// TIA Portal project "durum_grafigi_2_asansor" (V18)

(* hardware
DEVICE "S7-1200 station_1"  S7-1200 Station
   slot 0: "Rack_0"  S7-1200 Rack  Rack  V1.0
   slot 1: "PLC_1"  CPU 1214C DC/DC/DC  6ES7 214-1AG40-0XB0  V4.6
*)

// ===== PLC "PLC_1"  CPU 1214C DC/DC/DC =====

VAR_GLOBAL   // PLC tag table "Default tag table"
   "STOP-S0" AT %I0.0 : Bool;
   "START-S1" AT %I0.1 : Bool;
   "SAYMA SENSÖRÜ-S3" AT %I0.2 : Bool;
   "ASANSÖR AŞAĞIDA-S4" AT %I0.3 : Bool;
   "ASANSÖR YUKARIDA-S5" AT %I0.4 : Bool;
   "BANT MOTORU-M1" AT %Q0.0 : Bool;
   "ASANSÖR YUKARI-M2Y" AT %Q0.1 : Bool;
   "ASANSÖR AŞAĞI -M2A" AT %Q0.2 : Bool;
   "ASANSÖR KİLİTLEME" AT %Q0.3 : Bool;
   "PARÇA SÜRME" AT %Q0.4 : Bool;
   "DURUM_0 BAŞLANGIÇ" AT %M30.0 : Bool;
   "DURUM_1 BANT ÇALIŞTIRMA" AT %M30.1 : Bool;
   "DURUM_2 ASANSÖR YUKARI" AT %M30.2 : Bool;
   "DURUM_3 KİLİTLEME" AT %M30.3 : Bool;
   "DURUM_4 ASANSÖR AŞAĞI" AT %M30.4 : Bool;
   "System_Byte" AT %MB80 : Byte;
   "FirstScan" AT %M80.0 : Bool;
   "DiagStatusUpdate" AT %M80.1 : Bool;
   "AlwaysTRUE" AT %M80.2 : Bool;
   "AlwaysFALSE" AT %M80.3 : Bool;
   "Clock_Byte" AT %MB20 : Byte;
   "Clock_10Hz" AT %M20.0 : Bool;
   "Clock_5Hz" AT %M20.1 : Bool;
   "Clock_2.5Hz" AT %M20.2 : Bool;
   "Clock_2Hz" AT %M20.3 : Bool;
   "Clock_1.25Hz" AT %M20.4 : Bool;
   "Clock_1Hz" AT %M20.5 : Bool;
   "Clock_0.625Hz" AT %M20.6 : Bool;
   "Clock_0.5Hz" AT %M20.7 : Bool;
END_VAR

// folder: System blocks/Program resources

DATA_BLOCK "PARÇA SAYICISI"   // DB1
{ S7_Optimized_Access := 'TRUE' }
AUTHOR : Simatic
FAMILY : IEC
NAME : CNTR
VERSION : 1.0
// stored: InstanceOfName IEC_COUNTER
"IEC_COUNTER"
BEGIN
END_DATA_BLOCK

DATA_BLOCK "BEKLEME ZAMANI"   // DB2
{ S7_Optimized_Access := 'TRUE' }
AUTHOR : Simatic
FAMILY : IEC
NAME : IEC_TMR
VERSION : 1.0
// stored: InstanceOfName IEC_TIMER
"IEC_TIMER"
BEGIN
END_DATA_BLOCK

// folder: (top level)

ORGANIZATION_BLOCK "Main"   // OB1, LAD, ProgramCycle
TITLE = "Main Program Sweep (Cycle)"
{ S7_Optimized_Access := 'TRUE' }
VERSION : 0.1
// -*Asansör kabini asagida ve START butonuna basilmis ise
// bant dönmeye baslayacaktir.
// -*Bantin dönmeye baslamasiyla magazin üzerindeki
// paketler sürme silindiri yardimiyla belli araliklarla bant
// üzerine sürülecektir. Bant üzerindeki paketler SAYMA
// SENSÖRÜ önünden geçerek asansör kabinine dolacaktir.
// Kabin içerisindeki paket sayisi 5 oldugunda asansör
// yukan dogru hareket edecek ve bant duracaktir.
// -*Asansör kabini yukan çikip orada paketlerin bosalmasi
// için 5 saniye bekleyip tekrar asagi inecektir. Bekleme
// sirasinda FRENLEME çalisacaktir.
// -* START butonuna basildiginda bu islemler yeniden baslayacaktir.
// - STOP butonuna basildiginda FRENLEME çalisacak, diger motorlar duracaktir. STOP butonu
// birakildiginda BEKLEME SÜRESÌ tamamsa asansör asagi hareket edecektir.
   VAR_INPUT
      Initial_Call : Bool;   // Initial call of this OB
      Remanence : Bool;   // =True, if remanent data are available
   END_VAR
BEGIN

REGION Network 1: DURUM_0
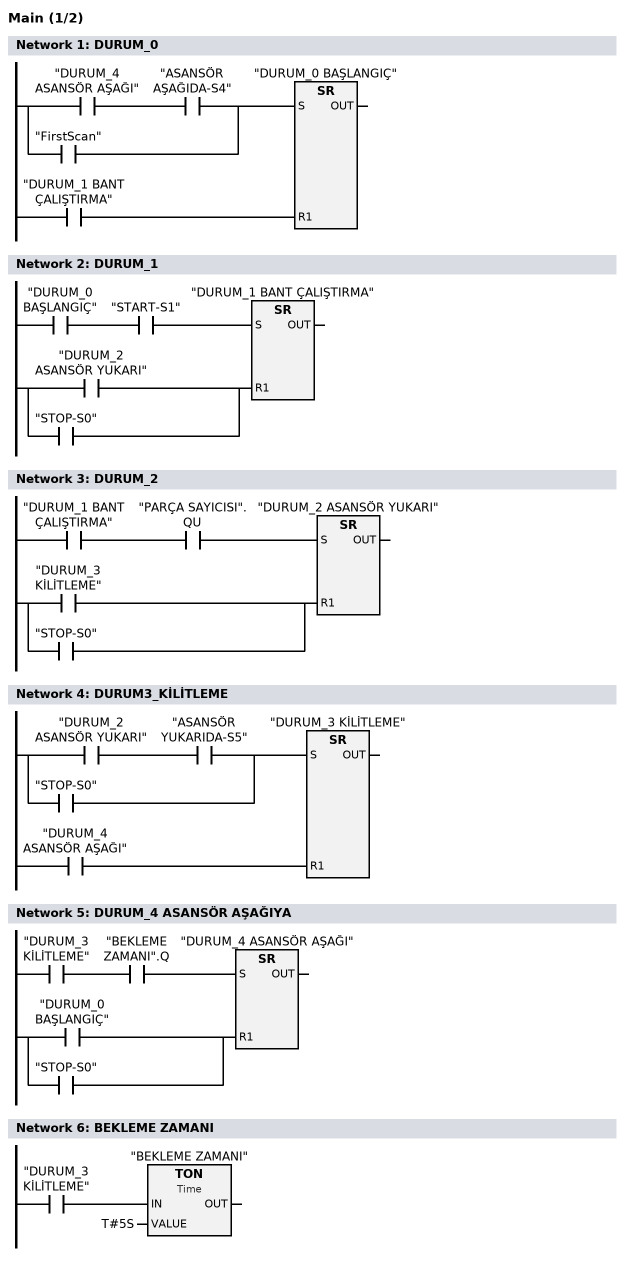
   RUNG wire#powerrail
      Contact( "DURUM_4 ASANSÖR AŞAĞI" )
      Contact( "ASANSÖR AŞAĞIDA-S4" )
      wire#w1
      S_SR(operand := "DURUM_0 BAŞLANGIÇ", r1 := wire#w2)
   END_RUNG
   RUNG wire#powerrail
      Contact( "FirstScan" )
   END_RUNG wire#w1
   RUNG wire#powerrail
      Contact( "DURUM_1 BANT ÇALIŞTIRMA" )
   END_RUNG wire#w2
   // the same network as SCL:
   IF ("DURUM_4 ASANSÖR AŞAĞI" AND "ASANSÖR AŞAĞIDA-S4") OR "FirstScan" THEN
       "DURUM_0 BAŞLANGIÇ" := TRUE;   // SR flip-flop
   END_IF;
   IF "DURUM_1 BANT ÇALIŞTIRMA" THEN "DURUM_0 BAŞLANGIÇ" := FALSE; END_IF;
END_REGION

REGION Network 2: DURUM_1
   RUNG wire#powerrail
      Contact( "DURUM_0 BAŞLANGIÇ" )
      Contact( "START-S1" )
      S_SR(operand := "DURUM_1 BANT ÇALIŞTIRMA", r1 := wire#w1)
   END_RUNG
   RUNG wire#powerrail
      Contact( "DURUM_2 ASANSÖR YUKARI" )
   END_RUNG wire#w1
   RUNG wire#powerrail
      Contact( "STOP-S0" )
   END_RUNG wire#w1
   // the same network as SCL:
   IF "DURUM_0 BAŞLANGIÇ" AND "START-S1" THEN
       "DURUM_1 BANT ÇALIŞTIRMA" := TRUE;   // SR flip-flop
   END_IF;
   IF "DURUM_2 ASANSÖR YUKARI" OR "STOP-S0" THEN "DURUM_1 BANT ÇALIŞTIRMA" := FALSE; END_IF;
END_REGION

REGION Network 3: DURUM_2
   RUNG wire#powerrail
      Contact( "DURUM_1 BANT ÇALIŞTIRMA" )
      Contact( "PARÇA SAYICISI".QU )
      S_SR(operand := "DURUM_2 ASANSÖR YUKARI", r1 := wire#w1)
   END_RUNG
   RUNG wire#powerrail
      Contact( "DURUM_3 KİLİTLEME" )
   END_RUNG wire#w1
   RUNG wire#powerrail
      Contact( "STOP-S0" )
   END_RUNG wire#w1
   // the same network as SCL:
   IF "DURUM_1 BANT ÇALIŞTIRMA" AND "PARÇA SAYICISI".QU THEN
       "DURUM_2 ASANSÖR YUKARI" := TRUE;   // SR flip-flop
   END_IF;
   IF "DURUM_3 KİLİTLEME" OR "STOP-S0" THEN "DURUM_2 ASANSÖR YUKARI" := FALSE; END_IF;
END_REGION

REGION Network 4: DURUM3_KİLİTLEME
   RUNG wire#powerrail
      Contact( "DURUM_2 ASANSÖR YUKARI" )
      Contact( "ASANSÖR YUKARIDA-S5" )
      wire#w1
      S_SR(operand := "DURUM_3 KİLİTLEME", r1 := wire#w2)
   END_RUNG
   RUNG wire#powerrail
      Contact( "STOP-S0" )
   END_RUNG wire#w1
   RUNG wire#powerrail
      Contact( "DURUM_4 ASANSÖR AŞAĞI" )
   END_RUNG wire#w2
   // the same network as SCL:
   IF ("DURUM_2 ASANSÖR YUKARI" AND "ASANSÖR YUKARIDA-S5") OR "STOP-S0" THEN
       "DURUM_3 KİLİTLEME" := TRUE;   // SR flip-flop
   END_IF;
   IF "DURUM_4 ASANSÖR AŞAĞI" THEN "DURUM_3 KİLİTLEME" := FALSE; END_IF;
END_REGION

REGION Network 5: DURUM_4 ASANSÖR AŞAĞIYA
   RUNG wire#powerrail
      Contact( "DURUM_3 KİLİTLEME" )
      Contact( "BEKLEME ZAMANI".Q )
      S_SR(operand := "DURUM_4 ASANSÖR AŞAĞI", r1 := wire#w1)
   END_RUNG
   RUNG wire#powerrail
      Contact( "DURUM_0 BAŞLANGIÇ" )
   END_RUNG wire#w1
   RUNG wire#powerrail
      Contact( "STOP-S0" )
   END_RUNG wire#w1
   // the same network as SCL:
   IF "DURUM_3 KİLİTLEME" AND "BEKLEME ZAMANI".Q THEN
       "DURUM_4 ASANSÖR AŞAĞI" := TRUE;   // SR flip-flop
   END_IF;
   IF "DURUM_0 BAŞLANGIÇ" OR "STOP-S0" THEN "DURUM_4 ASANSÖR AŞAĞI" := FALSE; END_IF;
END_REGION

REGION Network 6: BEKLEME ZAMANI
   "BEKLEME ZAMANI".TON(IN := "DURUM_3 KİLİTLEME", PT := T#5S);   // TON coil
END_REGION

REGION Network 7: SAYICI
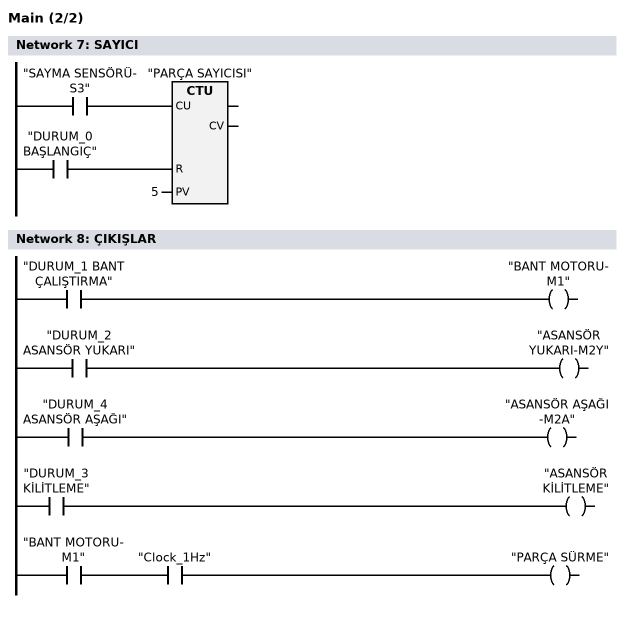
   "PARÇA SAYICISI".CTU(CU := "SAYMA SENSÖRÜ-S3", R := "DURUM_0 BAŞLANGIÇ", PV := 5);
END_REGION

REGION Network 8: ÇIKIŞLAR
   RUNG wire#powerrail
      Contact( "DURUM_1 BANT ÇALIŞTIRMA" )
      Coil( "BANT MOTORU-M1" )
   END_RUNG
   RUNG wire#powerrail
      Contact( "DURUM_2 ASANSÖR YUKARI" )
      Coil( "ASANSÖR YUKARI-M2Y" )
   END_RUNG
   RUNG wire#powerrail
      Contact( "DURUM_4 ASANSÖR AŞAĞI" )
      Coil( "ASANSÖR AŞAĞI -M2A" )
   END_RUNG
   RUNG wire#powerrail
      Contact( "DURUM_3 KİLİTLEME" )
      Coil( "ASANSÖR KİLİTLEME" )
   END_RUNG
   RUNG wire#powerrail
      Contact( "BANT MOTORU-M1" )
      Contact( "Clock_1Hz" )
      Coil( "PARÇA SÜRME" )
   END_RUNG
   // the same network as SCL:
   "BANT MOTORU-M1" := "DURUM_1 BANT ÇALIŞTIRMA";
   "ASANSÖR YUKARI-M2Y" := "DURUM_2 ASANSÖR YUKARI";
   "ASANSÖR AŞAĞI -M2A" := "DURUM_4 ASANSÖR AŞAĞI";
   "ASANSÖR KİLİTLEME" := "DURUM_3 KİLİTLEME";
   "PARÇA SÜRME" := "BANT MOTORU-M1" AND "Clock_1Hz";
END_REGION
END_ORGANIZATION_BLOCK